// SIMATIC S7-200 project (STEP 7-Micro/WIN), CPU 224XP CN REL 02.01

ORGANIZATION_BLOCK 主程序:OB1
TITLE=浙江天煌科技实业有限公司       http://www.tianhuang.cn          
// 创建人：十二车间售后组                                          
// 创建日期：2009.01.15                                                 
// 修改日期：2009.02.10       
//                                                                                                                                                                                   版本号：V1.1
BEGIN
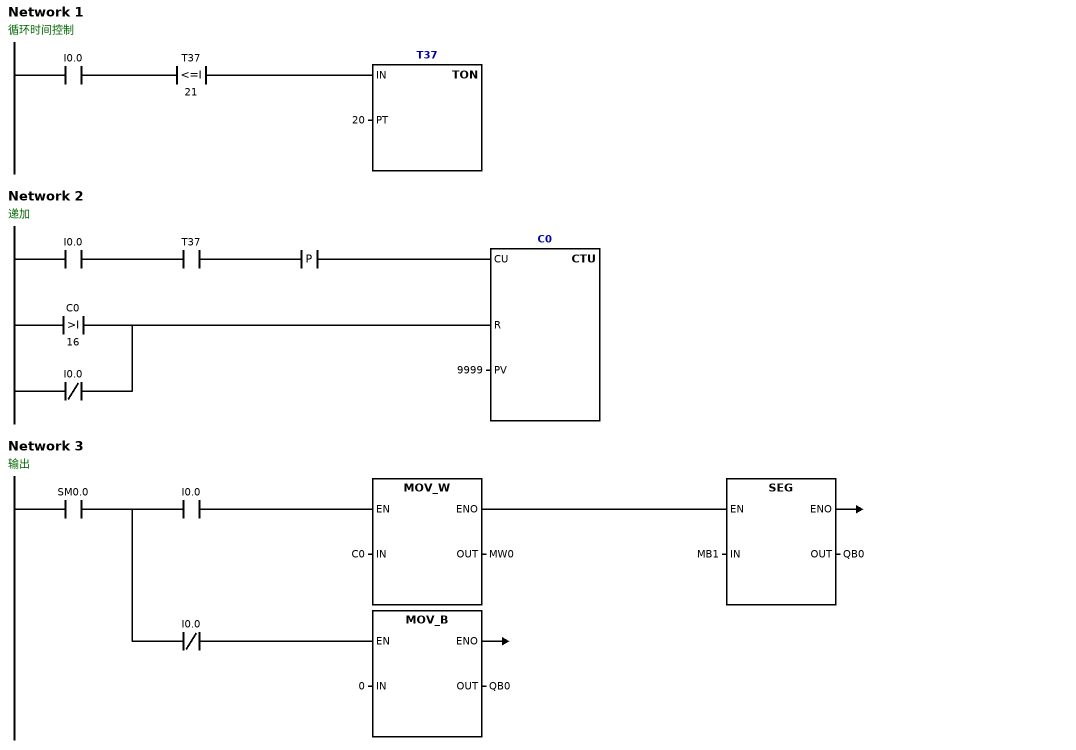
Network 1
// 循环时间控制
LD     I0.0
AW<=   T37, 21
TON    T37, 20
Network 2
// 递加
LD     I0.0
A      T37
EU
LDW>   C0, 16
ON     I0.0
CTU    C0, 9999
Network 3
// 输出
LD     SM0.0
LPS
A      I0.0
MOVW   C0, MW0
AENO
SEG    MB1, QB0
LPP
AN     I0.0
MOVB   0, QB0
END_ORGANIZATION_BLOCK
